FUNCTION_BLOCK FB_FastFaultLogger
VAR_INPUT
END_VAR
VAR_OUTPUT
END_VAR
VAR
END_VAR

END_FUNCTION_BLOCK

(* stored: Version 1.1.0.1, ProductVersion 3.1.4022.18
   POU FB_FastFaultLogger: Id {9c4f20b1-8d78-4ae8-9c90-0be1d68a7261}, SpecialFunc None *)
